(* Schneider Machine Expert - Basic project Lab-07-M221-autoOperator, file version 2.6.0.0 *)
(* ProjectInformations: Name=New project *)

HARDWARE
  Cpu 0: TM221ME16R/G
  ModuleExtensionObject 0: TM3DI8/G
  EthernetConfiguration: NetworkName=M221, IpAllocationMode=FixedAddress, IpAddress=0.0.0.0, SubnetMask=0.0.0.0
  SerialLineConfiguration: Baud=Baud19200, Parity=ParityEven, DataBits=DataBits8, StopBits=StopBits1, PhysicalMedium=PhysicalMediumRs485, TransmissionMode=TransmissionModeModbusRtu, SlaveId=1, Addressing=SlaveAddressing
  MastTask: UsePeriodScanMode=false, PeriodScan=100
  FastTask: Period=255
  CpuBehavior: StartingMode=StartAsPreviousState, AutoSaveRamOnEeprom=true, WatchdogPeriod=250

SYMBOLS  (address, symbol, comment, settings)
  %M0       ANYPOS
  %M1       MOVING
  %M2       ACC_IN_MANUAL
  %M3       ACC_IN_AUTO
  %M4       ACC_OUT_MANUAL
  %M5       ACC_OUT_AUTO
  %M6       NEW_POS
  %S13      SB_FIRSTRUN  "Indicates the first controller cycle in RUN mode"
  %MW0      PCR
  %MW1      POS
  %MW2      TARGET_POS
  %MW10     TMPW
  %MW11     POS_BUFF
  %MW20     LEN
  %TM0      ACC_DELAY  [Preset=2, Base=OneSecond]
  %TM1      DEC_DELAY  [Type=TOF, Preset=2, Base=OneSecond]
  %C0       STEPS  [Preset=0]
  %I0.0     AUTO
  %I0.1     DL1
  %I0.2     DL2
  %I0.3     DL3
  %I0.4     DL4
  %I0.5     DL5
  %I0.6     BTN_FW
  %I0.7     BTN_RV
  %Q0.0     FW
  %Q0.1     RV
  %Q0.2     SPD
  %I1.0     BTN_STOP

POU Generic functions
  (* SectionNumber=1 *)

// Rung 0
// Load distance list
  LD %S13                 (* SB_FIRSTRUN *)
  [ %MW20 := 5 ]          (* LEN *)
  [ %MW21 := 3 ]
  [ %MW22 := 4 ]
  [ %MW23 := 2 ]
  // as ST:
  //   IF SB_FIRSTRUN THEN LEN := 5; END_IF;
  //   IF SB_FIRSTRUN THEN %MW21 := 3; END_IF;
  //   IF SB_FIRSTRUN THEN %MW22 := 4; END_IF;
  //   IF SB_FIRSTRUN THEN %MW23 := 2; END_IF;

// Rung 1
// Detect any postiton
  LD %I0.1                (* DL1 *)
  OR %I0.2                (* DL2 *)
  OR %I0.3                (* DL3 *)
  OR %I0.4                (* DL4 *)
  OR %I0.5                (* DL5 *)
  ST %M0                  (* ANYPOS *)
  // as ST:
  //   ANYPOS := DL1 OR DL2 OR DL3 OR DL4 OR DL5;

// Rung 2
// Position detection - cyclic method init
  LDR %M0                 (* ANYPOS *)
  [ %MW11 := %I0.0:8 ]    (* POS_BUFF, AUTO *)
  [ %MW11 := SHR ( %MW11 AND 16#003E , 1 ) ](* POS_BUFF, POS_BUFF *)
  [ %MW1 := 0 ]           (* POS *)
  // as ST:
  //   IF RISING(ANYPOS) THEN POS_BUFF := AUTO:8; END_IF;
  //   IF RISING(ANYPOS) THEN POS_BUFF := SHR ( POS_BUFF AND 16#003E , 1 ); END_IF;
  //   IF RISING(ANYPOS) THEN POS := 0; END_IF;

// Rung 3 %L0
// Position detection - cyclic method loop
  %L0:
  LD %M0                  (* ANYPOS *)
  AND [ %MW11 > 0 ]       (* POS_BUFF *)
  [ INC %MW1 ]            (* POS *)
  [ %MW11 := SHR ( %MW11 , 1 ) ](* POS_BUFF, POS_BUFF *)
  JMPC %L0
  // as ST:
  //   %L0:
  //   IF ANYPOS AND POS_BUFF > 0 THEN INC POS; END_IF;
  //   _t1 := ANYPOS AND POS_BUFF > 0;
  //   IF _t1 THEN POS_BUFF := SHR ( POS_BUFF , 1 ); END_IF;
  //   IF _t1 THEN JMP %L0; END_IF;

// Rung 4
// Detect moving
  LD %Q0.0                (* FW *)
  OR %Q0.1                (* RV *)
  ST %M1                  (* MOVING *)
  // as ST:
  //   MOVING := FW OR RV;

// Rung 5
// Acceleration delay input
  LD %I0.0                (* AUTO *)
  AND %M3                 (* ACC_IN_AUTO *)
  OR(N %I0.0              (* AUTO *)
  AND %M2                 (* ACC_IN_MANUAL *)
  )
  IN %TM0                 (* ACC_DELAY *)
  // as ST:
  //   ACC_DELAY(IN := AUTO AND ACC_IN_AUTO OR NOT AUTO AND ACC_IN_MANUAL);

// Rung 6
// Acceleration delay output
  LD %M5                  (* ACC_OUT_AUTO *)
  OR %M4                  (* ACC_OUT_MANUAL *)
  ST %Q0.2                (* SPD *)
  // as ST:
  //   SPD := ACC_OUT_AUTO OR ACC_OUT_MANUAL;

// Rung 7
// Emergency stop
  LDR %I1.0               (* BTN_STOP *)
  SR0
  // as ST:
  //   IF RISING(BTN_STOP) THEN SR0(); END_IF;

POU Manual mode
  (* SectionNumber=2 *)

// Rung 8
// Manual - stop
  LDN %I0.0               (* AUTO *)
  AND( %Q0.0              (* FW *)
  AND(N %I0.6             (* BTN_FW *)
  OR %I0.5                (* DL5 *)
  )
  OR( %Q0.1               (* RV *)
  AND(N %I0.7             (* BTN_RV *)
  OR %I0.1                (* DL1 *)
  )
  )
  )
  ANDR %M0                (* ANYPOS *)
  SR0                     (* STOP *)
  // as ST:
  //   IF NOT AUTO AND (FW AND (NOT BTN_FW OR DL5) OR RV AND (NOT BTN_RV OR DL1)) AND RISING(ANYPOS) THEN SR0(); END_IF;

// Rung 9
// Manual - start forward
  LDN %I0.0               (* AUTO *)
  ANDR %I0.6              (* BTN_FW *)
  ANDN %I0.5              (* DL5 *)
  S %Q0.0                 (* FW *)
  // as ST:
  //   IF NOT AUTO AND RISING(BTN_FW) AND NOT DL5 THEN FW := TRUE; END_IF;

// Rung 10
// Manual - start backward
  LDN %I0.0               (* AUTO *)
  ANDR %I0.7              (* BTN_RV *)
  ANDN %I0.1              (* DL1 *)
  S %Q0.1                 (* RV *)
  // as ST:
  //   IF NOT AUTO AND RISING(BTN_RV) AND NOT DL1 THEN RV := TRUE; END_IF;

// Rung 11
// Manual - acceleration delay
  LDN %I0.0               (* AUTO *)
  AND( %Q0.0              (* FW *)
  AND %I0.6               (* BTN_FW *)
  )
  OR( %Q0.1               (* RV *)
  AND %I0.7               (* BTN_RV *)
  )
  ST %M2                  (* ACC_IN_MANUAL *)
  // as ST:
  //   ACC_IN_MANUAL := NOT AUTO AND FW AND BTN_FW OR RV AND BTN_RV;

// Rung 12
// Manual - acceleration
  LDN %I0.0               (* AUTO *)
  AND %TM0.Q              (* ACC_DELAY *)
  ST %M4                  (* ACC_OUT_MANUAL *)
  // as ST:
  //   ACC_OUT_MANUAL := NOT AUTO AND ACC_DELAY.Q;

POU Auto mode
  (* SectionNumber=3 *)

// Rung 13
// Auto - new target position
  LD %I0.0                (* AUTO *)
  AND [ %MW0 > 0 ]        (* PCR *)
  AND [ %MW2 = 0 ]        (* TARGET_POS *)
  ST %M6                  (* NEW_POS *)
  // as ST:
  //   NEW_POS := AUTO AND PCR > 0 AND TARGET_POS = 0;

// Rung 14
// Auto - target position equal to current
  IF0
  AND %M6                 (* NEW_POS *)
  AND [ %MW0 = %MW1 ]     (* PCR, POS *)
  THEN0

// Rung 15
// Auto - abort movig
  [ %MW0 := 0 ]           (* PCR *)
  // as ST:
  //   PCR := 0;

// Rung 16
// Auto - start moving
  ELSE0
  AND %M6                 (* NEW_POS *)
  MPS
  [ %MW2 := %MW0 ]        (* TARGET_POS, PCR *)
  [ %MW10 := LW ( ABS ( DWORD ( %MW2 - %MW1 ) ) ) ](* TMPW, TARGET_POS, POS *)
  [ %C0.P := %MW10 ]      (* STEPS, TMPW *)
  S %C0                   (* STEPS *)
  [ %MW10 := %MW2 - 2 ]   (* TMPW, TARGET_POS *)
  MRD
  AND [ %MW2 > %MW1 ]     (* TARGET_POS, POS *)
  [ %TM1.P := %MW20[%MW10] ](* DEC_DELAY, LEN, TMPW *)
  S %Q0.0                 (* FW *)
  MPP
  AND [ %MW2 < %MW1 ]     (* TARGET_POS, POS *)
  [ INC %MW10 ]           (* TMPW *)
  [ %TM1.P := %MW20[%MW10] ](* DEC_DELAY, LEN, TMPW *)
  S %Q0.1                 (* RV *)

// Rung 17
// Auto - start condition end
  ENDIF0

// Rung 18
// Auto - acceleration/deceleration delay
  LD %I0.0                (* AUTO *)
  AND %M1                 (* MOVING *)
  MPS
  ST %M3                  (* ACC_IN_AUTO *)
  MPP
  AND [ %C0.V > 0 ]       (* STEPS *)
  IN %TM1                 (* DEC_DELAY *)
  // as ST:
  //   ACC_IN_AUTO := AUTO AND MOVING;
  //   DEC_DELAY(IN := AUTO AND MOVING AND STEPS.V > 0);

// Rung 19
// Auto - steps count
  LD %I0.0                (* AUTO *)
  AND %M1                 (* MOVING *)
  ANDF %M0                (* ANYPOS *)
  AND [ %C0.V > 0 ]       (* STEPS *)
  CD %C0                  (* STEPS *)
  // as ST:
  //   STEPS(CD := AUTO AND MOVING AND FALLING(ANYPOS) AND STEPS.V > 0);

// Rung 20
// Auto - acceleration
  LD %I0.0                (* AUTO *)
  AND %TM0.Q              (* ACC_DELAY *)
  AND %TM1.Q              (* DEC_DELAY *)
  ST %M5                  (* ACC_OUT_AUTO *)
  // as ST:
  //   ACC_OUT_AUTO := AUTO AND ACC_DELAY.Q AND DEC_DELAY.Q;

// Rung 21
// Auto - stop
  LD %I0.0                (* AUTO *)
  AND %M1                 (* MOVING *)
  AND %M0                 (* ANYPOS *)
  AND [ %MW2 = %MW1 ]     (* TARGET_POS, POS *)
  SR0                     (* STOP *)
  [ %MW2 := 0 ]           (* TARGET_POS *)
  [ %MW0 := 0 ]           (* PCR *)
  // as ST:
  //   IF AUTO AND MOVING AND ANYPOS AND TARGET_POS = POS THEN SR0(); END_IF;
  //   _t1 := AUTO AND MOVING AND ANYPOS AND TARGET_POS = POS;
  //   IF _t1 THEN TARGET_POS := 0; END_IF;
  //   IF _t1 THEN PCR := 0; END_IF;

Subroutine STOP
  (* SectionNumber=4, Number=0 *)

// Rung 22
// Stop moving
  LD 1
  R %Q0.0                 (* FW *)
  R %Q0.1                 (* RV *)
  R %Q0.2                 (* SPD *)
  // as ST:
  //   FW := FALSE;
  //   RV := FALSE;
  //   SPD := FALSE;
